// TIA Portal V19 export
DATA_BLOCK "TDISCON_DI"   // DB368
// stored: AutoNumber false, InstanceOfName T_DISCON, OfSystemLibElement TDISCON, OfSystemLibVersion 2.1
"T_DISCON"
   // VAR_INPUT
   //    REQ : Bool := FALSE;
   //    ID : CONN_OUC := 16#0000;
   // END_VAR
   // VAR_OUTPUT
   //    DONE : Bool := FALSE;
   //    BUSY : Bool := FALSE;
   //    ERROR : Bool := FALSE;
   //    STATUS : Word := 16#7000;
   // END_VAR
BEGIN
END_DATA_BLOCK
